INTERFACE I_AlarmManager

// Acknowledges all uacknowledged alarms.
METHOD AcknowledgeAllAlarms
END_METHOD

// Provides access to action builder with fluent approach.
METHOD PUBLIC Actions : I_AlarmActions
VAR_INPUT
END_VAR
END_METHOD

{attribute 'monitoring':='call'}
// Gets the total count of currently active alarms
PROPERTY ActiveAlarmsCount : UINT
GET
END_GET
END_PROPERTY

// Deletes the alarm with the provided id.
METHOD DeleteAlarm
VAR_INPUT
	id	: DINT;
END_VAR
END_METHOD

// Deletes all existing alarms from the memory
METHOD DeleteAll
END_METHOD

{attribute 'monitoring':='call'}
// Gets or sets if alarm manager is enabled or not. When disabled, all active alarms will become inactive!
PROPERTY Enable : BOOL
GET
END_GET
SET
END_SET
END_PROPERTY

(* Gets the alarm with the provided id. 
 If no mathching alarm exists, an invalid reference will be returned - check by using __ISVALIDREF() for any further operations!.*)
METHOD GetAlarmById : REFERENCE TO ST_AlarmInfo
VAR_INPUT
	nID		: T_ArrayIndexer;	// Id of the alarm.
END_VAR
END_METHOD

// Gets the alarm with the provided name. 
// IF no mathching alarm exists, an invalid REFERENCE will be returned - check BY using __ISVALIDREF() FOR ANY further operations!.*)
METHOD GetAlarmByName : REFERENCE TO ST_AlarmInfo
VAR_INPUT
	sName	: Tc2_System.T_MaxString;	// Name of the alarm
END_VAR
END_METHOD

// Registers a new alarm with the provided information. 
// Returns TRUE if new alarm was registered or false if not
// Possible reasons for fail:
// - alarm buffer is full
// - the id already exists)
METHOD RegisterAlarm : BOOL
VAR_INPUT
	Id		: T_ArrayIndexer;			// Alarm ID
	Name	: Tc2_System.T_MaxString;	// Alarm name
	Message	: Tc2_System.T_MaxString;	// Message when the alarm occurrs
	Level	: E_AlarmLevel;				// Alarm level
END_VAR
END_METHOD

{attribute 'monitoring':='call'}
// Gets the total number of alarms registered
PROPERTY RegisteredAlarmsCount : UDINT
GET
END_GET
END_PROPERTY

{attribute 'monitoring':='call'}
// Gets the current count of alarms that have not yet been acknowledged
PROPERTY UnacknowledgedAlarmsCount : UINT
GET
END_GET
END_PROPERTY

END_INTERFACE

(* stored: Version 1.1.0.1
   Itf I_AlarmManager: Id {08ed33cf-534a-0dd0-0916-694bc76d6975}
   Method AcknowledgeAllAlarms: Id {1e530507-ece4-0bf2-30ca-7dc1ee9b6502}
   Method Actions: Id {7fd5adb5-f699-0d3c-28ab-9bbe59531087}
   Property ActiveAlarmsCount: Id {2d6bf4ab-360d-092e-201b-11f8e5f47030}
   Get Get: Id {ed5d2186-6859-0c04-1ea3-b4f44ecf585c}
   Method DeleteAlarm: Id {a7a177eb-524a-0c9a-1c86-c39a7191d952}
   Method DeleteAll: Id {4c68625a-8348-0ede-3967-a08de81c0997}
   Property Enable: Id {0ae510b3-be57-0ba1-3645-7ca74f263283}
   Get Get: Id {d641b5cb-4afe-06fc-37fc-e223f0c5a6b9}
   Set Set: Id {767625c3-1355-05c7-1af5-5dda3ede591a}
   Method GetAlarmById: Id {6794a080-844b-0a8a-010d-0b8faf92f607}
   Method GetAlarmByName: Id {b6a13b3a-4fe4-05b4-03de-e547fbc7db95}
   Method RegisterAlarm: Id {7b9e25e7-d788-0c73-0fbd-360da521ec34}
   Property RegisteredAlarmsCount: Id {b79b6ee5-f1af-0dc0-1ef4-907a3b0ef213}
   Get Get: Id {175362fc-405e-0254-3605-0a7d81ea3e6b}
   Property UnacknowledgedAlarmsCount: Id {565ebd05-d113-0bc4-354e-0d80b658fc2f}
   Get Get: Id {44ad48c8-561a-014b-1364-bd809079d93f} *)
